FUNCTION_BLOCK FB_UdintTrig
VAR_INPUT
	uiIn:UDINT;
END_VAR
VAR_OUTPUT
	bOut: BOOL;

END_VAR
VAR
	uiOld:UDINT;
	tAllowNewErr:TON;
	bFirst:BOOL:=TRUE;
END_VAR


bOut:= uiIn <> uiOld AND tAllowNewErr.Q AND NOT bFirst;
tAllowNewErr(IN:=uiIn = uiOld , PT:= T#5S);
uiOld:=uiIn;
bFirst:=FALSE;

END_FUNCTION_BLOCK

(* stored: Version 1.1.0.1, ProductVersion 3.1.4024.4
   POU FB_UdintTrig: Id {fc5fcc48-b681-4638-be88-fc6128cbbdae}, SpecialFunc None *)
